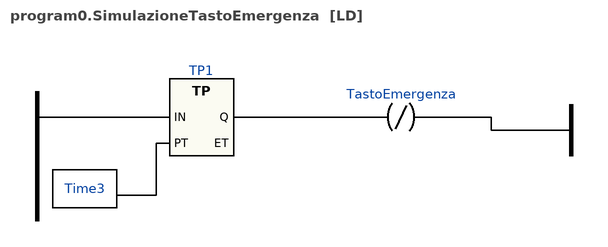
(* [picture p24: program0.SimulazioneTastoEmergenza, LD] *)
(* LD diagram, written out as Structured Text *)
TP1(IN := TRUE, PT := Time3);
TastoEmergenza := NOT TP1.Q;
END_ACTION

ACTION SimulazioneTastoCaricaBusta:
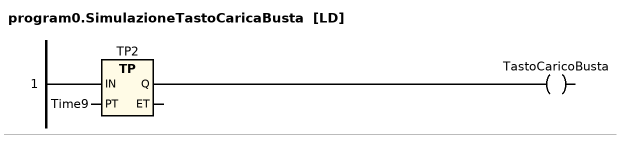
(* LD diagram, written out as Structured Text *)
TP2(IN := TRUE, PT := Time9);
TastoCaricoBusta := TP2.Q;
END_ACTION
END_PROGRAM

CONFIGURATION Config0
  RESOURCE Res0 ON PLC
    TASK task0(INTERVAL := T#20ms, PRIORITY := 0);
    PROGRAM instance0 WITH task0 : program0;
  END_RESOURCE
END_CONFIGURATION
